// TIA Portal V17 export
// export: Created 2025-03-10T12:17:47.1815291Z, ExportSetting WithDefaults, DisplayName Totally Integrated Automation Portal, DisplayVersion V17 Update 8, DisplayName TIA Portal Openness, DisplayVersion V17 Update 8, DisplayName TIA Portal Version Control Interface, DisplayVersion V17, DisplayName SINAMICS Startdrive Advanced, DisplayVersion V17 SP2, DisplayName SINAMICS Startdrive G110M, G120, G120C, G120D, G120P, G115D, DisplayVersion V17 SP2, DisplayName SINAMICS Startdrive G130, G150, S120, S150, SINAMICS MV, S210, DisplayVersion V17 SP2, DisplayName STEP 7 Professional, DisplayVersion V17 Update 8, DisplayName SINUMERIK ONE STEP 7 Toolbox, DisplayVersion V17 Update 12, DisplayName SINUMERIK 840D sl STEP 7 Toolbox, DisplayVersion V17 Update 12, DisplayName STEP 7 Safety, DisplayVersion V17 Update 6, DisplayName WinCC Advanced, DisplayVersion V17 Update 8
TYPE "LBP_typeModularMcpUniversalInput"
TITLE = Modular MCP image / Imagen de MCP modulares / Abbild modulare MCP
// Input image of universal keypad for modular MCP / Imagen de entrada del panel de mando universal de MCP modulares / Eingangsabbild des Universal-Bedienfelds für modulare MCP
// stored: IsFailsafeCompliant false
   STRUCT
      key0 : Bool;   // Eingangsabbild n+0 Bit 0 / input image n+0 bit 0 / Imagen de entrada n+0 bit 0
      key1 : Bool;   // Eingangsabbild n+0 Bit 1 / input image n+0 bit 1 / Imagen de entrada n+0 bit 1
      key2 : Bool;   // Eingangsabbild n+0 Bit 2 / input image n+0 bit 2 / Imagen de entrada n+0 bit 2
      key3 : Bool;   // Eingangsabbild n+0 Bit 3 / input image n+0 bit 3 / Imagen de entrada n+0 bit 3
      key4 : Bool;   // Eingangsabbild n+0 Bit 4 / input image n+0 bit 4 / Imagen de entrada n+0 bit 4
      key5 : Bool;   // Eingangsabbild n+0 Bit 5 / input image n+0 bit 5 / Imagen de entrada n+0 bit 5
      key6 : Bool;   // Eingangsabbild n+0 Bit 6 / input image n+0 bit 6 / Imagen de entrada n+0 bit 6
      key7 : Bool;   // Eingangsabbild n+0 Bit 7 / input image n+0 bit 7 / Imagen de entrada n+0 bit 7
      key8 : Bool;   // Eingangsabbild n+1 Bit 0 / input image n+1 bit 0 / Imagen de entrada n+1 bit 0
      key9 : Bool;   // Eingangsabbild n+1 Bit 1 / input image n+1 bit 1 / Imagen de entrada n+1 bit 1
      key10 : Bool;   // Eingangsabbild n+1 Bit 2 / input image n+1 bit 2 / Imagen de entrada n+1 bit 2
      key11 : Bool;   // Eingangsabbild n+1 Bit 3 / input image n+1 bit 3 / Imagen de entrada n+1 bit 3
      key12 : Bool;   // Eingangsabbild n+1 Bit 4 / input image n+1 bit 4 / Imagen de entrada n+1 bit 4
      key13 : Bool;   // Eingangsabbild n+1 Bit 5 / input image n+1 bit 5 / Imagen de entrada n+1 bit 5
      key14 : Bool;   // Eingangsabbild n+1 Bit 6 / input image n+1 bit 6 / Imagen de entrada n+1 bit 6
      reserved17 : Bool;
      key16 : Bool;   // Eingangsabbild n+2 Bit 0 / input image n+2 bit 0 / Imagen de entrada n+2 bit 0
      key17 : Bool;   // Eingangsabbild n+2 Bit 1 / input image n+2 bit 1 / Imagen de entrada n+2 bit 1
      key18 : Bool;   // Eingangsabbild n+2 Bit 2 / input image n+2 bit 2 / Imagen de entrada n+2 bit 2
      reserved23 : Bool;
      reserved24 : Bool;
      reserved25 : Bool;
      reserved26 : Bool;
      reserved27 : Bool;
      key24 : Bool;   // Eingangsabbild n+3 Bit 0 / input image n+3 bit 0 / Imagen de entrada n+3 bit 0
      key25 : Bool;   // Eingangsabbild n+3 Bit 1 / input image n+3 bit 1 / Imagen de entrada n+3 bit 1
      key26 : Bool;   // Eingangsabbild n+3 Bit 2 / input image n+3 bit 2 / Imagen de entrada n+3 bit 2
      reserved33 : Bool;
      reserved34 : Bool;
      reserved35 : Bool;
      reserved36 : Bool;
      reserved37 : Bool;
   END_STRUCT;
END_TYPE
